// Mitsubishi GX Works2 project: fx3g程序模板   PLC: FX3G

PROGRAM MAIN
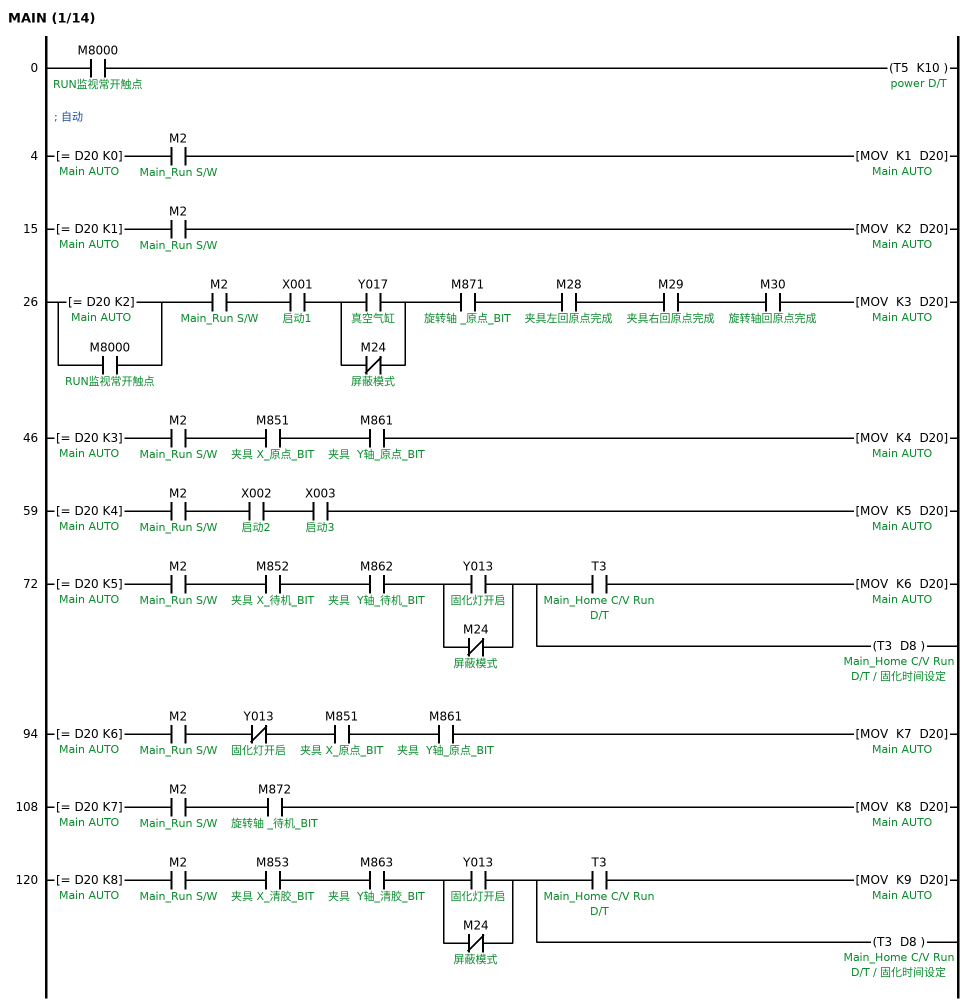
0     LD      M8000  ; RUN监视常开触点
      OUT     T5 K10  ; power D/T
; 自动
4     LD=     D20 K0  ; Main AUTO
      AND     M2  ; Main_Run S/W
      MOV     K1 D20
15    LD=     D20 K1  ; Main AUTO
      AND     M2  ; Main_Run S/W
      MOV     K2 D20
26    LD=     D20 K2  ; Main AUTO
      OR      M8000  ; RUN监视常开触点
      AND     M2  ; Main_Run S/W
      AND     X001  ; 启动1
      LD      Y017  ; 真空气缸
      ORI     M24  ; 屏蔽模式
      ANB
      AND     M871  ; 旋转轴 _原点_BIT
      AND     M28  ; 夹具左回原点完成
      AND     M29  ; 夹具右回原点完成
      AND     M30  ; 旋转轴回原点完成
      MOV     K3 D20
46    LD=     D20 K3  ; Main AUTO
      AND     M2  ; Main_Run S/W
      AND     M851  ; 夹具 X_原点_BIT
      AND     M861  ; 夹具  Y轴_原点_BIT
      MOV     K4 D20
59    LD=     D20 K4  ; Main AUTO
      AND     M2  ; Main_Run S/W
      AND     X002  ; 启动2
      AND     X003  ; 启动3
      MOV     K5 D20
72    LD=     D20 K5  ; Main AUTO
      AND     M2  ; Main_Run S/W
      AND     M852  ; 夹具 X_待机_BIT
      AND     M862  ; 夹具  Y轴_待机_BIT
      LD      Y013  ; 固化灯开启
      ORI     M24  ; 屏蔽模式
      ANB
      MPS
      AND     T3  ; Main_Home C/V Run D/T
      MOV     K6 D20
      MPP
      OUT     T3 D8  ; Main_Home C/V Run D/T / 固化时间设定
94    LD=     D20 K6  ; Main AUTO
      AND     M2  ; Main_Run S/W
      ANI     Y013  ; 固化灯开启
      AND     M851  ; 夹具 X_原点_BIT
      AND     M861  ; 夹具  Y轴_原点_BIT
      MOV     K7 D20
108   LD=     D20 K7  ; Main AUTO
      AND     M2  ; Main_Run S/W
      AND     M872  ; 旋转轴 _待机_BIT
      MOV     K8 D20
120   LD=     D20 K8  ; Main AUTO
      AND     M2  ; Main_Run S/W
      AND     M853  ; 夹具 X_清胶_BIT
      AND     M863  ; 夹具  Y轴_清胶_BIT
      LD      Y013  ; 固化灯开启
      ORI     M24  ; 屏蔽模式
      ANB
      MPS
      AND     T3  ; Main_Home C/V Run D/T
      MOV     K9 D20
      MPP
      OUT     T3 D8  ; Main_Home C/V Run D/T / 固化时间设定
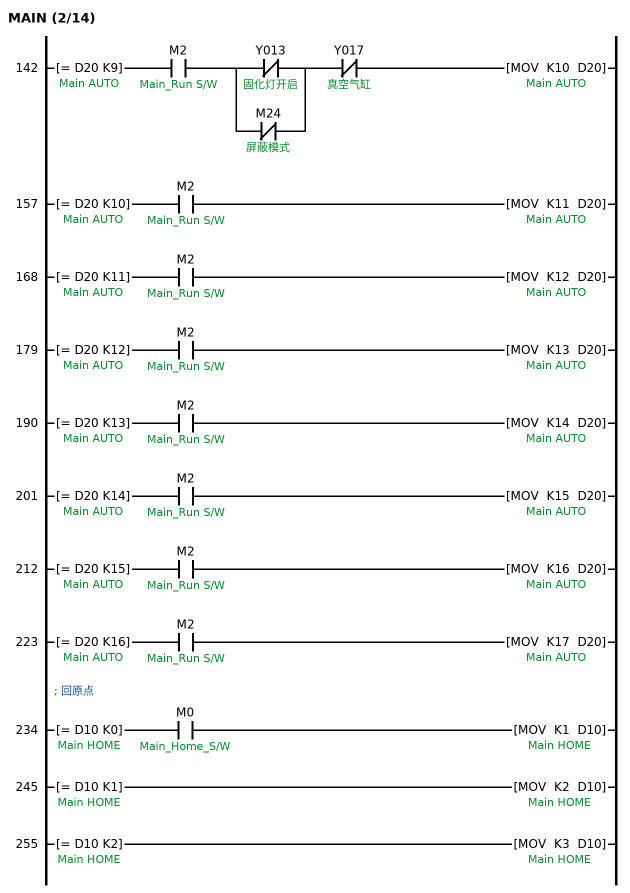
142   LD=     D20 K9  ; Main AUTO
      AND     M2  ; Main_Run S/W
      LDI     Y013  ; 固化灯开启
      ORI     M24  ; 屏蔽模式
      ANB
      ANI     Y017  ; 真空气缸
      MOV     K10 D20
157   LD=     D20 K10  ; Main AUTO
      AND     M2  ; Main_Run S/W
      MOV     K11 D20
168   LD=     D20 K11  ; Main AUTO
      AND     M2  ; Main_Run S/W
      MOV     K12 D20
179   LD=     D20 K12  ; Main AUTO
      AND     M2  ; Main_Run S/W
      MOV     K13 D20
190   LD=     D20 K13  ; Main AUTO
      AND     M2  ; Main_Run S/W
      MOV     K14 D20
201   LD=     D20 K14  ; Main AUTO
      AND     M2  ; Main_Run S/W
      MOV     K15 D20
212   LD=     D20 K15  ; Main AUTO
      AND     M2  ; Main_Run S/W
      MOV     K16 D20
223   LD=     D20 K16  ; Main AUTO
      AND     M2  ; Main_Run S/W
      MOV     K17 D20
; 回原点
234   LD=     D10 K0  ; Main HOME
      AND     M0  ; Main_Home_S/W
      MOV     K1 D10
245   LD=     D10 K1  ; Main HOME
      MOV     K2 D10
255   LD=     D10 K2  ; Main HOME
      MOV     K3 D10
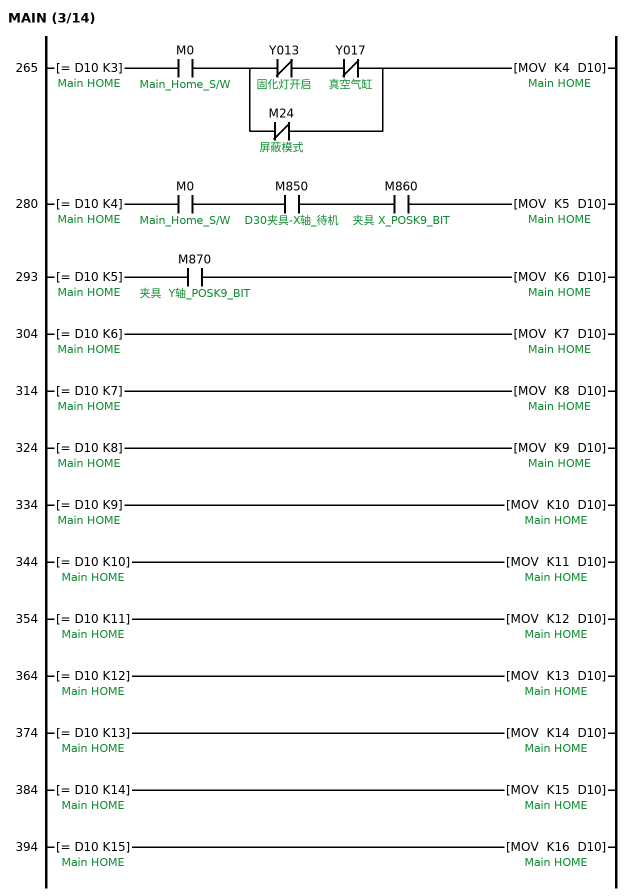
265   LD=     D10 K3  ; Main HOME
      AND     M0  ; Main_Home_S/W
      LDI     Y013  ; 固化灯开启
      ANI     Y017  ; 真空气缸
      ORI     M24  ; 屏蔽模式
      ANB
      MOV     K4 D10
280   LD=     D10 K4  ; Main HOME
      AND     M0  ; Main_Home_S/W
      AND     M850  ; D30夹具-X轴_待机
      AND     M860  ; 夹具 X_POSK9_BIT
      MOV     K5 D10
293   LD=     D10 K5  ; Main HOME
      AND     M870  ; 夹具  Y轴_POSK9_BIT
      MOV     K6 D10
304   LD=     D10 K6  ; Main HOME
      MOV     K7 D10
314   LD=     D10 K7  ; Main HOME
      MOV     K8 D10
324   LD=     D10 K8  ; Main HOME
      MOV     K9 D10
334   LD=     D10 K9  ; Main HOME
      MOV     K10 D10
344   LD=     D10 K10  ; Main HOME
      MOV     K11 D10
354   LD=     D10 K11  ; Main HOME
      MOV     K12 D10
364   LD=     D10 K12  ; Main HOME
      MOV     K13 D10
374   LD=     D10 K13  ; Main HOME
      MOV     K14 D10
384   LD=     D10 K14  ; Main HOME
      MOV     K15 D10
394   LD=     D10 K15  ; Main HOME
      MOV     K16 D10
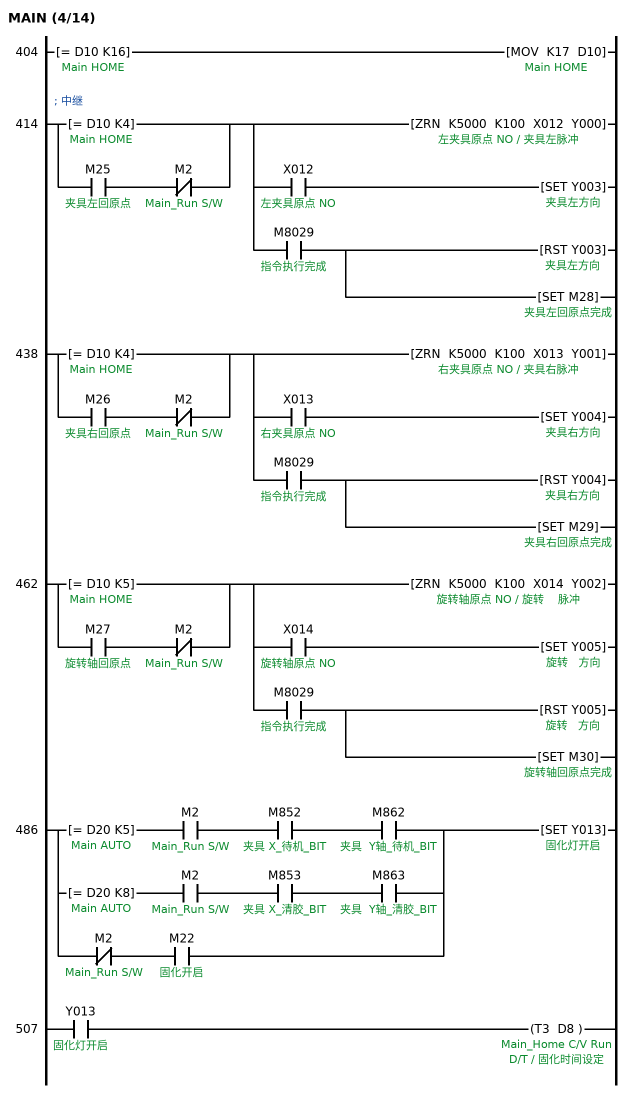
404   LD=     D10 K16  ; Main HOME
      MOV     K17 D10
; 中继
414   LD=     D10 K4  ; Main HOME
      LD      M25  ; 夹具左回原点
      ANI     M2  ; Main_Run S/W
      ORB
      ZRN     K5000 K100 X012 Y000  ; 左夹具原点 NO / 夹具左脉冲
      MPS
      AND     X012  ; 左夹具原点 NO
      SET     Y003  ; 夹具左方向
      MPP
      AND     M8029  ; 指令执行完成
      RST     Y003  ; 夹具左方向
      SET     M28  ; 夹具左回原点完成
438   LD=     D10 K4  ; Main HOME
      LD      M26  ; 夹具右回原点
      ANI     M2  ; Main_Run S/W
      ORB
      ZRN     K5000 K100 X013 Y001  ; 右夹具原点 NO / 夹具右脉冲
      MPS
      AND     X013  ; 右夹具原点 NO
      SET     Y004  ; 夹具右方向
      MPP
      AND     M8029  ; 指令执行完成
      RST     Y004  ; 夹具右方向
      SET     M29  ; 夹具右回原点完成
462   LD=     D10 K5  ; Main HOME
      LD      M27  ; 旋转轴回原点
      ANI     M2  ; Main_Run S/W
      ORB
      ZRN     K5000 K100 X014 Y002  ; 旋转轴原点 NO / 旋转    脉冲
      MPS
      AND     X014  ; 旋转轴原点 NO
      SET     Y005  ; 旋转   方向
      MPP
      AND     M8029  ; 指令执行完成
      RST     Y005  ; 旋转   方向
      SET     M30  ; 旋转轴回原点完成
486   LD=     D20 K5  ; Main AUTO
      AND     M2  ; Main_Run S/W
      AND     M852  ; 夹具 X_待机_BIT
      AND     M862  ; 夹具  Y轴_待机_BIT
      LD=     D20 K8  ; Main AUTO
      AND     M2  ; Main_Run S/W
      AND     M853  ; 夹具 X_清胶_BIT
      AND     M863  ; 夹具  Y轴_清胶_BIT
      ORB
      LDI     M2  ; Main_Run S/W
      AND     M22  ; 固化开启
      ORB
      SET     Y013  ; 固化灯开启
507   LD      Y013  ; 固化灯开启
      OUT     T3 D8  ; Main_Home C/V Run D/T / 固化时间设定
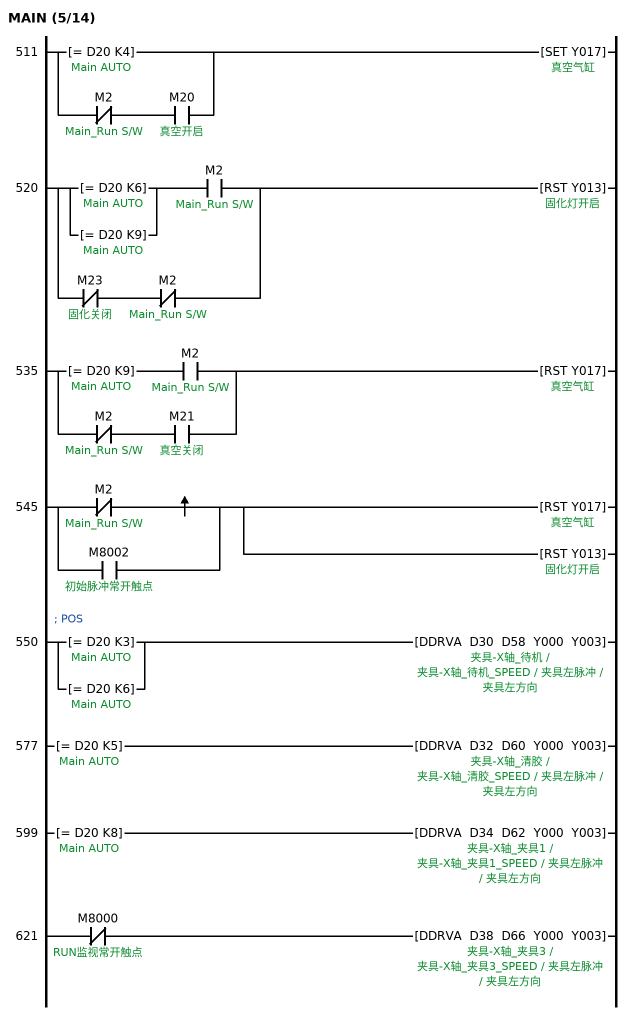
511   LD=     D20 K4  ; Main AUTO
      LDI     M2  ; Main_Run S/W
      AND     M20  ; 真空开启
      ORB
      SET     Y017  ; 真空气缸
520   LD=     D20 K6  ; Main AUTO
      OR=     D20 K9  ; Main AUTO
      AND     M2  ; Main_Run S/W
      LDI     M23  ; 固化关闭
      ANI     M2  ; Main_Run S/W
      ORB
      RST     Y013  ; 固化灯开启
535   LD=     D20 K9  ; Main AUTO
      AND     M2  ; Main_Run S/W
      LDI     M2  ; Main_Run S/W
      AND     M21  ; 真空关闭
      ORB
      RST     Y017  ; 真空气缸
545   LDI     M2  ; Main_Run S/W
      MEP
      OR      M8002  ; 初始脉冲常开触点
      RST     Y017  ; 真空气缸
      RST     Y013  ; 固化灯开启
; POS
550   LD=     D20 K3  ; Main AUTO
      OR=     D20 K6  ; Main AUTO
      DDRVA   D30 D58 Y000 Y003  ; 夹具-X轴_待机 / 夹具-X轴_待机_SPEED
577   LD=     D20 K5  ; Main AUTO
      DDRVA   D32 D60 Y000 Y003  ; 夹具-X轴_清胶 / 夹具-X轴_清胶_SPEED
599   LD=     D20 K8  ; Main AUTO
      DDRVA   D34 D62 Y000 Y003  ; 夹具-X轴_夹具1 / 夹具-X轴_夹具1_SPEED
621   LDI     M8000  ; RUN监视常开触点
      DDRVA   D38 D66 Y000 Y003  ; 夹具-X轴_夹具3 / 夹具-X轴_夹具3_SPEED
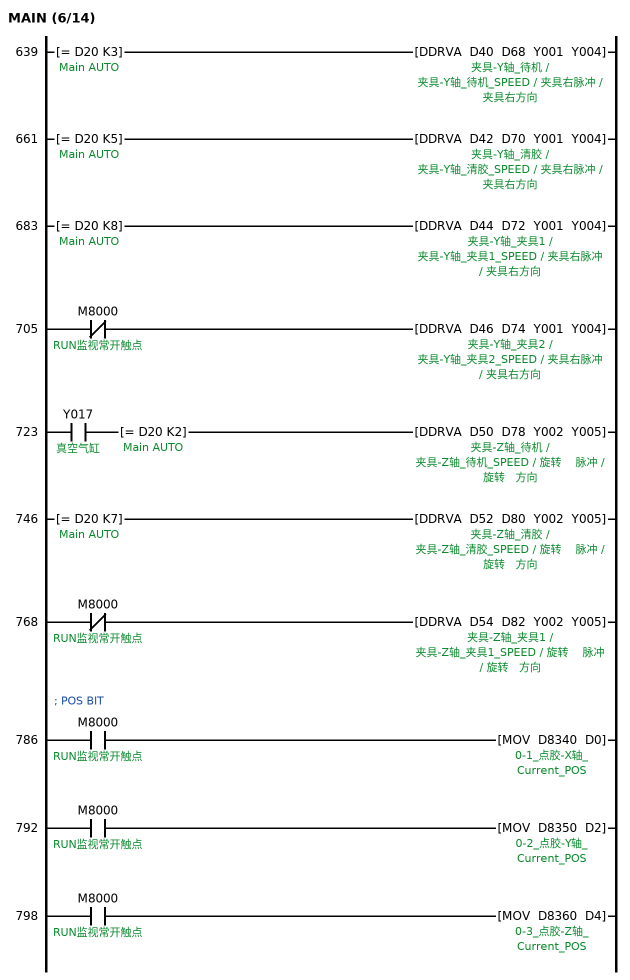
639   LD=     D20 K3  ; Main AUTO
      DDRVA   D40 D68 Y001 Y004  ; 夹具-Y轴_待机 / 夹具-Y轴_待机_SPEED
661   LD=     D20 K5  ; Main AUTO
      DDRVA   D42 D70 Y001 Y004  ; 夹具-Y轴_清胶 / 夹具-Y轴_清胶_SPEED
683   LD=     D20 K8  ; Main AUTO
      DDRVA   D44 D72 Y001 Y004  ; 夹具-Y轴_夹具1 / 夹具-Y轴_夹具1_SPEED
705   LDI     M8000  ; RUN监视常开触点
      DDRVA   D46 D74 Y001 Y004  ; 夹具-Y轴_夹具2 / 夹具-Y轴_夹具2_SPEED
723   LD      Y017  ; 真空气缸
      AND=    D20 K2  ; Main AUTO
      DDRVA   D50 D78 Y002 Y005  ; 夹具-Z轴_待机 / 夹具-Z轴_待机_SPEED
746   LD=     D20 K7  ; Main AUTO
      DDRVA   D52 D80 Y002 Y005  ; 夹具-Z轴_清胶 / 夹具-Z轴_清胶_SPEED
768   LDI     M8000  ; RUN监视常开触点
      DDRVA   D54 D82 Y002 Y005  ; 夹具-Z轴_夹具1 / 夹具-Z轴_夹具1_SPEED
; POS BIT
786   LD      M8000  ; RUN监视常开触点
      MOV     D8340 D0  ; 0-1_点胶-X轴_Current_POS
792   LD      M8000  ; RUN监视常开触点
      MOV     D8350 D2  ; 0-2_点胶-Y轴_Current_POS
798   LD      M8000  ; RUN监视常开触点
      MOV     D8360 D4  ; 0-3_点胶-Z轴_Current_POS
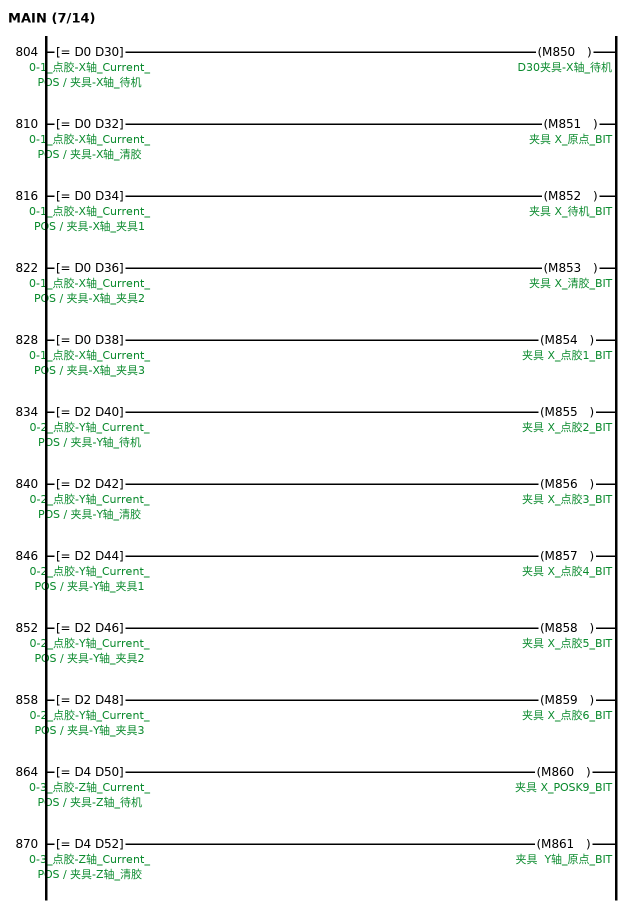
804   LD=     D0 D30  ; 0-1_点胶-X轴_Current_POS / 夹具-X轴_待机
      OUT     M850  ; D30夹具-X轴_待机
810   LD=     D0 D32  ; 0-1_点胶-X轴_Current_POS / 夹具-X轴_清胶
      OUT     M851  ; 夹具 X_原点_BIT
816   LD=     D0 D34  ; 0-1_点胶-X轴_Current_POS / 夹具-X轴_夹具1
      OUT     M852  ; 夹具 X_待机_BIT
822   LD=     D0 D36  ; 0-1_点胶-X轴_Current_POS / 夹具-X轴_夹具2
      OUT     M853  ; 夹具 X_清胶_BIT
828   LD=     D0 D38  ; 0-1_点胶-X轴_Current_POS / 夹具-X轴_夹具3
      OUT     M854  ; 夹具 X_点胶1_BIT
834   LD=     D2 D40  ; 0-2_点胶-Y轴_Current_POS / 夹具-Y轴_待机
      OUT     M855  ; 夹具 X_点胶2_BIT
840   LD=     D2 D42  ; 0-2_点胶-Y轴_Current_POS / 夹具-Y轴_清胶
      OUT     M856  ; 夹具 X_点胶3_BIT
846   LD=     D2 D44  ; 0-2_点胶-Y轴_Current_POS / 夹具-Y轴_夹具1
      OUT     M857  ; 夹具 X_点胶4_BIT
852   LD=     D2 D46  ; 0-2_点胶-Y轴_Current_POS / 夹具-Y轴_夹具2
      OUT     M858  ; 夹具 X_点胶5_BIT
858   LD=     D2 D48  ; 0-2_点胶-Y轴_Current_POS / 夹具-Y轴_夹具3
      OUT     M859  ; 夹具 X_点胶6_BIT
864   LD=     D4 D50  ; 0-3_点胶-Z轴_Current_POS / 夹具-Z轴_待机
      OUT     M860  ; 夹具 X_POSK9_BIT
870   LD=     D4 D52  ; 0-3_点胶-Z轴_Current_POS / 夹具-Z轴_清胶
      OUT     M861  ; 夹具  Y轴_原点_BIT
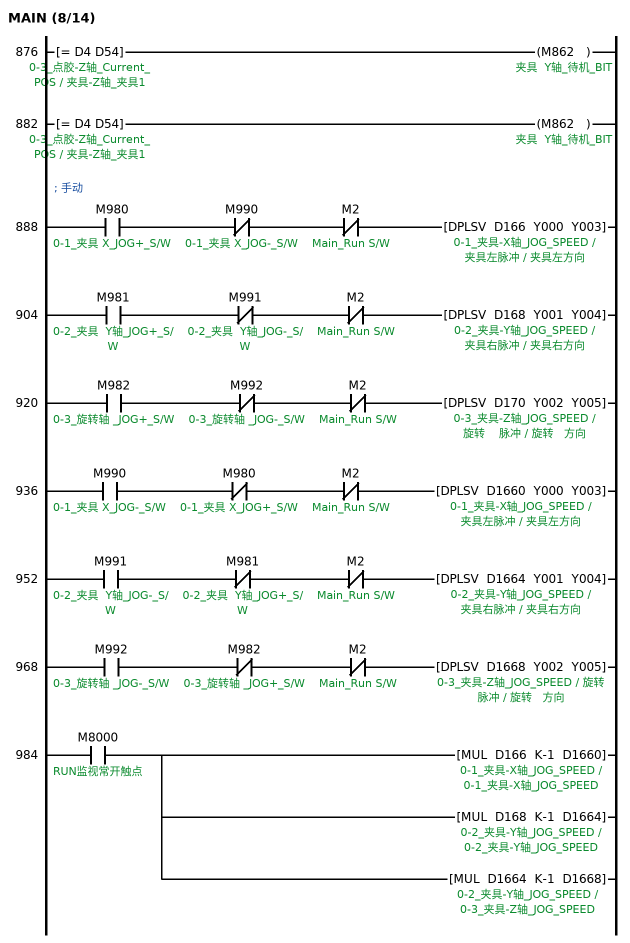
876   LD=     D4 D54  ; 0-3_点胶-Z轴_Current_POS / 夹具-Z轴_夹具1
      OUT     M862  ; 夹具  Y轴_待机_BIT
882   LD=     D4 D54  ; 0-3_点胶-Z轴_Current_POS / 夹具-Z轴_夹具1
      OUT     M862  ; 夹具  Y轴_待机_BIT
; 手动
888   LD      M980  ; 0-1_夹具 X_JOG+_S/W
      ANI     M990  ; 0-1_夹具 X_JOG-_S/W
      ANI     M2  ; Main_Run S/W
      DPLSV   D166 Y000 Y003  ; 0-1_夹具-X轴_JOG_SPEED
904   LD      M981  ; 0-2_夹具  Y轴_JOG+_S/W
      ANI     M991  ; 0-2_夹具  Y轴_JOG-_S/W
      ANI     M2  ; Main_Run S/W
      DPLSV   D168 Y001 Y004  ; 0-2_夹具-Y轴_JOG_SPEED
920   LD      M982  ; 0-3_旋转轴 _JOG+_S/W
      ANI     M992  ; 0-3_旋转轴 _JOG-_S/W
      ANI     M2  ; Main_Run S/W
      DPLSV   D170 Y002 Y005  ; 0-3_夹具-Z轴_JOG_SPEED
936   LD      M990  ; 0-1_夹具 X_JOG-_S/W
      ANI     M980  ; 0-1_夹具 X_JOG+_S/W
      ANI     M2  ; Main_Run S/W
      DPLSV   D1660 Y000 Y003  ; 0-1_夹具-X轴_JOG_SPEED
952   LD      M991  ; 0-2_夹具  Y轴_JOG-_S/W
      ANI     M981  ; 0-2_夹具  Y轴_JOG+_S/W
      ANI     M2  ; Main_Run S/W
      DPLSV   D1664 Y001 Y004  ; 0-2_夹具-Y轴_JOG_SPEED
968   LD      M992  ; 0-3_旋转轴 _JOG-_S/W
      ANI     M982  ; 0-3_旋转轴 _JOG+_S/W
      ANI     M2  ; Main_Run S/W
      DPLSV   D1668 Y002 Y005  ; 0-3_夹具-Z轴_JOG_SPEED
984   LD      M8000  ; RUN监视常开触点
      MUL     D166 K-1 D1660
      MUL     D168 K-1 D1664
      MUL     D1664 K-1 D1668
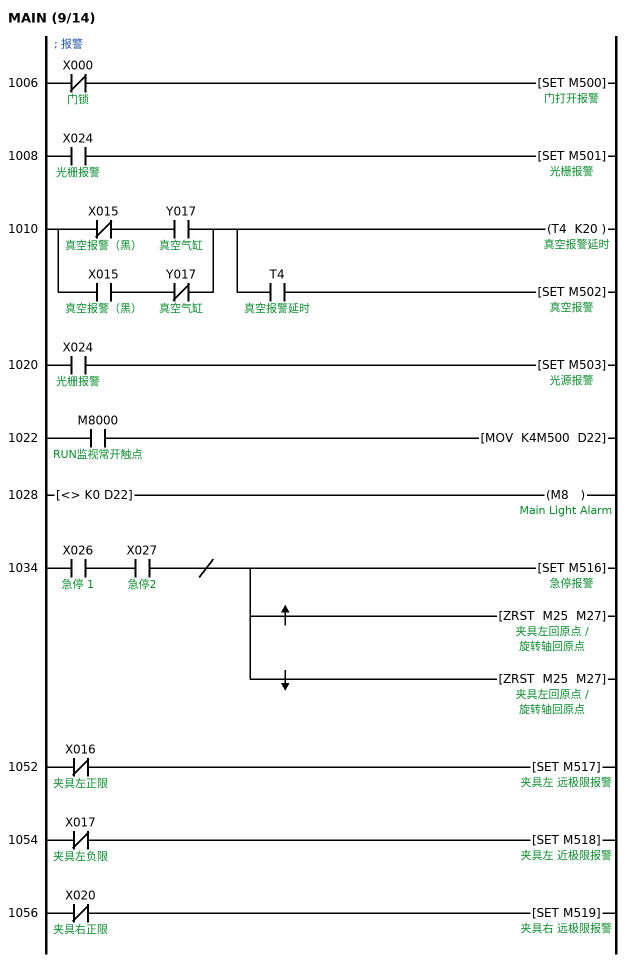
; 报警
1006  LDI     X000  ; 门锁
      SET     M500  ; 门打开报警
1008  LD      X024  ; 光栅报警
      SET     M501  ; 光栅报警
1010  LDI     X015  ; 真空报警（黑）
      AND     Y017  ; 真空气缸
      LD      X015  ; 真空报警（黑）
      ANI     Y017  ; 真空气缸
      ORB
      OUT     T4 K20  ; 真空报警延时
      AND     T4  ; 真空报警延时
      SET     M502  ; 真空报警
1020  LD      X024  ; 光栅报警
      SET     M503  ; 光源报警
1022  LD      M8000  ; RUN监视常开触点
      MOV     K4M500 D22
1028  LD<>    K0 D22
      OUT     M8  ; Main Light Alarm
1034  LD      X026  ; 急停 1
      AND     X027  ; 急停2
      INV
      SET     M516  ; 急停报警
      MPS
      MEP
      ZRST    M25 M27
      MPP
      MEF
      ZRST    M25 M27
1052  LDI     X016  ; 夹具左正限
      SET     M517  ; 夹具左 远极限报警
1054  LDI     X017  ; 夹具左负限
      SET     M518  ; 夹具左 近极限报警
1056  LDI     X020  ; 夹具右正限
      SET     M519  ; 夹具右 远极限报警
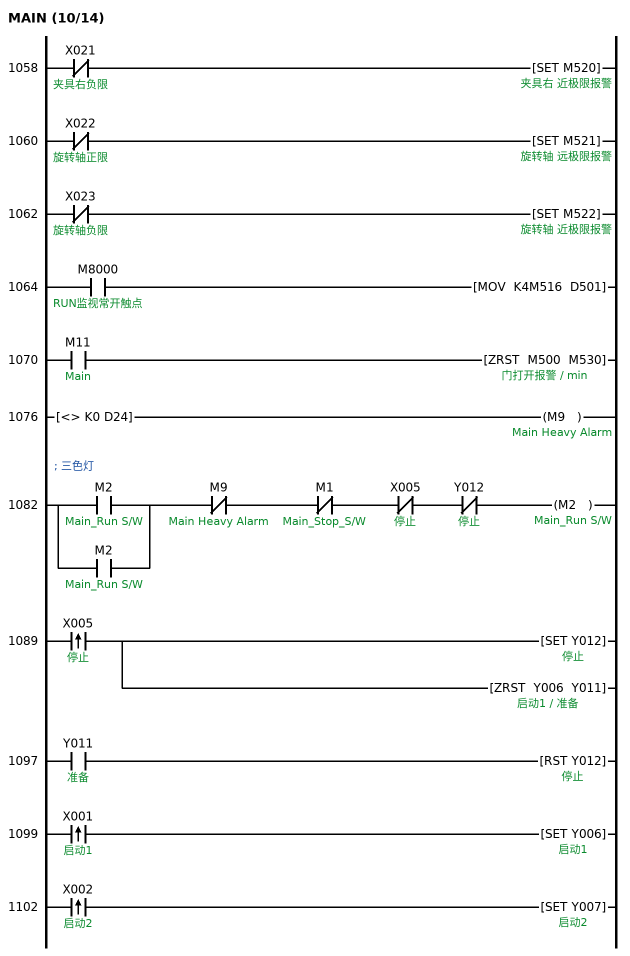
1058  LDI     X021  ; 夹具右负限
      SET     M520  ; 夹具右 近极限报警
1060  LDI     X022  ; 旋转轴正限
      SET     M521  ; 旋转轴 远极限报警
1062  LDI     X023  ; 旋转轴负限
      SET     M522  ; 旋转轴 近极限报警
1064  LD      M8000  ; RUN监视常开触点
      MOV     K4M516 D501
1070  LD      M11  ; Main
      ZRST    M500 M530  ; min
1076  LD<>    K0 D24
      OUT     M9  ; Main Heavy Alarm
; 三色灯
1082  LD      M2  ; Main_Run S/W
      OR      M2  ; Main_Run S/W
      ANI     M9  ; Main Heavy Alarm
      ANI     M1  ; Main_Stop_S/W
      ANI     X005  ; 停止
      ANI     Y012  ; 停止
      OUT     M2  ; Main_Run S/W
1089  LDP     X005  ; 停止
      SET     Y012  ; 停止
      ZRST    Y006 Y011  ; 启动1 / 准备
1097  LD      Y011  ; 准备
      RST     Y012  ; 停止
1099  LDP     X001  ; 启动1
      SET     Y006  ; 启动1
1102  LDP     X002  ; 启动2
      SET     Y007  ; 启动2
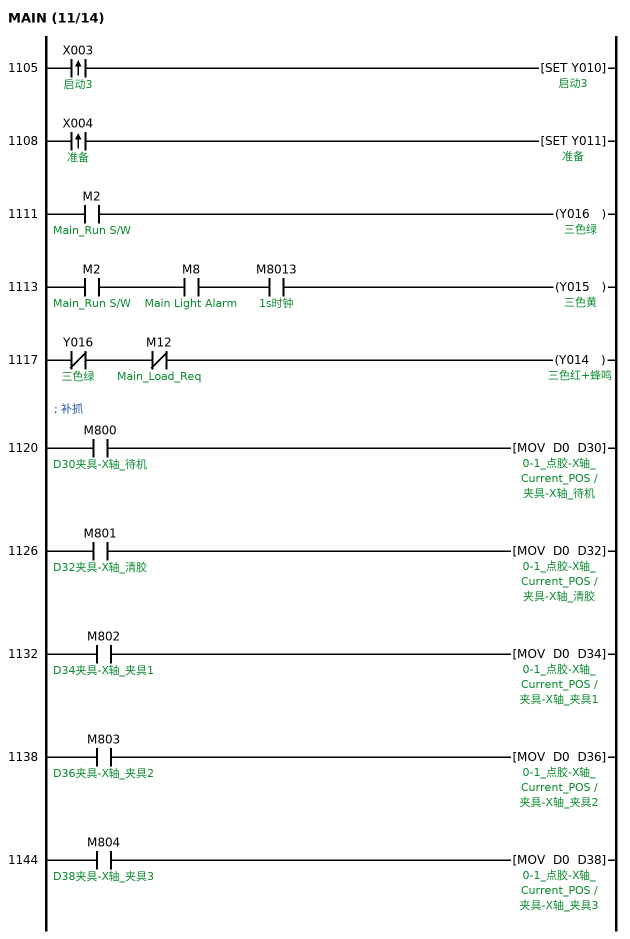
1105  LDP     X003  ; 启动3
      SET     Y010  ; 启动3
1108  LDP     X004  ; 准备
      SET     Y011  ; 准备
1111  LD      M2  ; Main_Run S/W
      OUT     Y016  ; 三色绿
1113  LD      M2  ; Main_Run S/W
      AND     M8  ; Main Light Alarm
      AND     M8013  ; 1s时钟
      OUT     Y015  ; 三色黄
1117  LDI     Y016  ; 三色绿
      ANI     M12  ; Main_Load_Req
      OUT     Y014  ; 三色红+蜂鸣
; 补抓
1120  LD      M800  ; D30夹具-X轴_待机
      MOV     D0 D30
1126  LD      M801  ; D32夹具-X轴_清胶
      MOV     D0 D32
1132  LD      M802  ; D34夹具-X轴_夹具1
      MOV     D0 D34
1138  LD      M803  ; D36夹具-X轴_夹具2
      MOV     D0 D36
1144  LD      M804  ; D38夹具-X轴_夹具3
      MOV     D0 D38
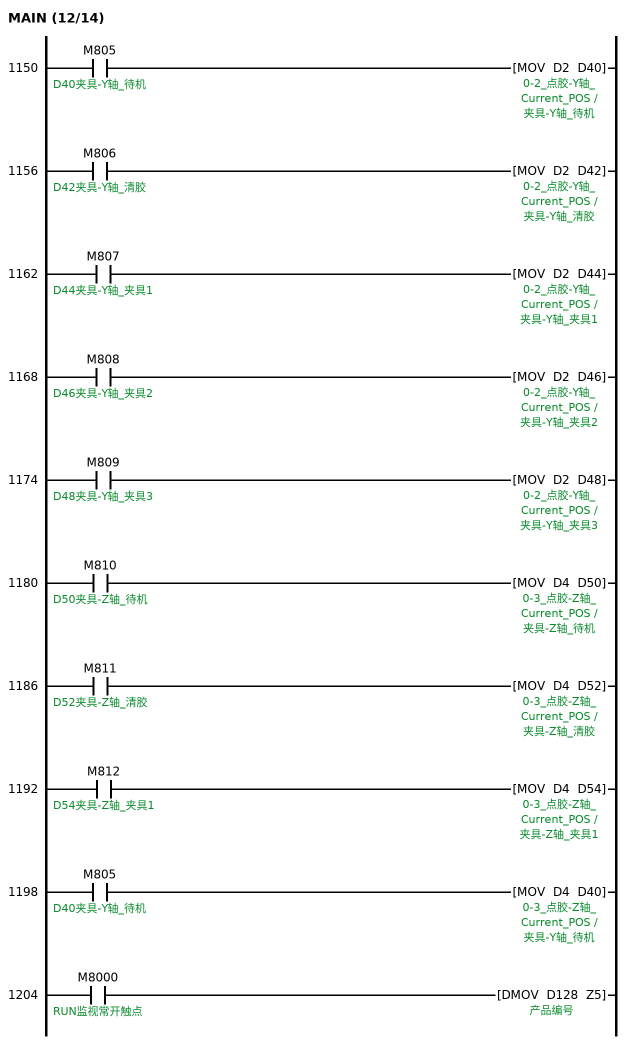
1150  LD      M805  ; D40夹具-Y轴_待机
      MOV     D2 D40
1156  LD      M806  ; D42夹具-Y轴_清胶
      MOV     D2 D42
1162  LD      M807  ; D44夹具-Y轴_夹具1
      MOV     D2 D44
1168  LD      M808  ; D46夹具-Y轴_夹具2
      MOV     D2 D46
1174  LD      M809  ; D48夹具-Y轴_夹具3
      MOV     D2 D48
1180  LD      M810  ; D50夹具-Z轴_待机
      MOV     D4 D50
1186  LD      M811  ; D52夹具-Z轴_清胶
      MOV     D4 D52
1192  LD      M812  ; D54夹具-Z轴_夹具1
      MOV     D4 D54
1198  LD      M805  ; D40夹具-Y轴_待机
      MOV     D4 D40
1204  LD      M8000  ; RUN监视常开触点
      DMOV    D128 Z5  ; 产品编号
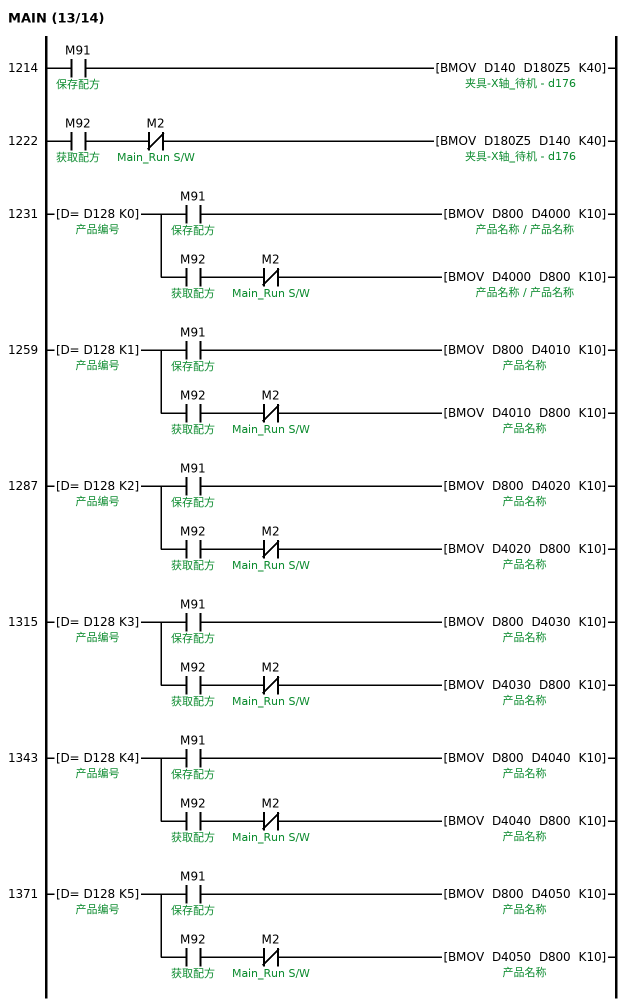
1214  LD      M91  ; 保存配方
      BMOV    D140 D180Z5 K40  ; 夹具-X轴_待机 - d176
1222  LD      M92  ; 获取配方
      ANI     M2  ; Main_Run S/W
      BMOV    D180Z5 D140 K40
1231  LDD=    D128 K0  ; 产品编号
      MPS
      AND     M91  ; 保存配方
      BMOV    D800 D4000 K10  ; 产品名称 / 产品名称
      MPP
      AND     M92  ; 获取配方
      ANI     M2  ; Main_Run S/W
      BMOV    D4000 D800 K10
1259  LDD=    D128 K1  ; 产品编号
      MPS
      AND     M91  ; 保存配方
      BMOV    D800 D4010 K10
      MPP
      AND     M92  ; 获取配方
      ANI     M2  ; Main_Run S/W
      BMOV    D4010 D800 K10
1287  LDD=    D128 K2  ; 产品编号
      MPS
      AND     M91  ; 保存配方
      BMOV    D800 D4020 K10
      MPP
      AND     M92  ; 获取配方
      ANI     M2  ; Main_Run S/W
      BMOV    D4020 D800 K10
1315  LDD=    D128 K3  ; 产品编号
      MPS
      AND     M91  ; 保存配方
      BMOV    D800 D4030 K10
      MPP
      AND     M92  ; 获取配方
      ANI     M2  ; Main_Run S/W
      BMOV    D4030 D800 K10
1343  LDD=    D128 K4  ; 产品编号
      MPS
      AND     M91  ; 保存配方
      BMOV    D800 D4040 K10
      MPP
      AND     M92  ; 获取配方
      ANI     M2  ; Main_Run S/W
      BMOV    D4040 D800 K10
1371  LDD=    D128 K5  ; 产品编号
      MPS
      AND     M91  ; 保存配方
      BMOV    D800 D4050 K10
      MPP
      AND     M92  ; 获取配方
      ANI     M2  ; Main_Run S/W
      BMOV    D4050 D800 K10
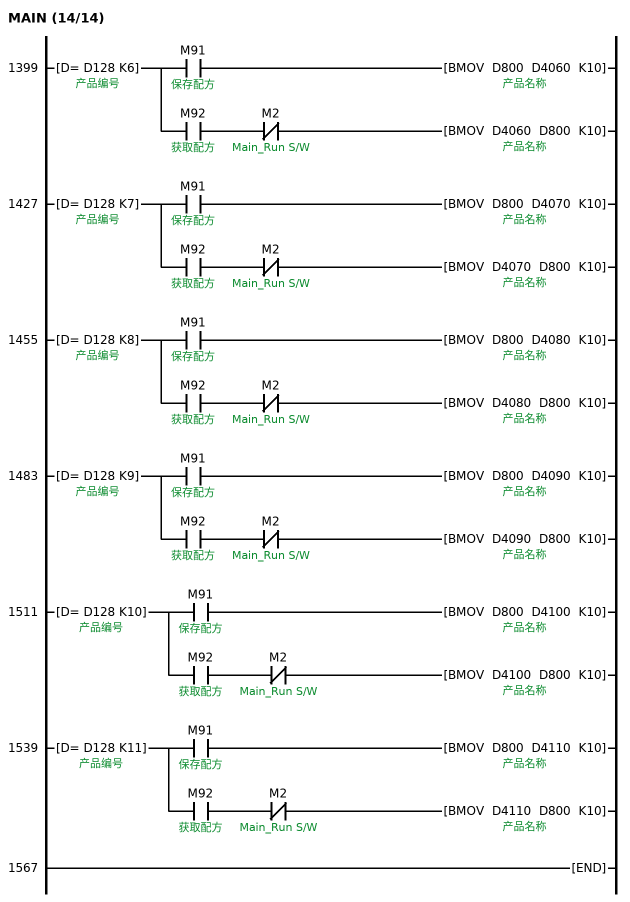
1399  LDD=    D128 K6  ; 产品编号
      MPS
      AND     M91  ; 保存配方
      BMOV    D800 D4060 K10
      MPP
      AND     M92  ; 获取配方
      ANI     M2  ; Main_Run S/W
      BMOV    D4060 D800 K10
1427  LDD=    D128 K7  ; 产品编号
      MPS
      AND     M91  ; 保存配方
      BMOV    D800 D4070 K10
      MPP
      AND     M92  ; 获取配方
      ANI     M2  ; Main_Run S/W
      BMOV    D4070 D800 K10
1455  LDD=    D128 K8  ; 产品编号
      MPS
      AND     M91  ; 保存配方
      BMOV    D800 D4080 K10
      MPP
      AND     M92  ; 获取配方
      ANI     M2  ; Main_Run S/W
      BMOV    D4080 D800 K10
1483  LDD=    D128 K9  ; 产品编号
      MPS
      AND     M91  ; 保存配方
      BMOV    D800 D4090 K10
      MPP
      AND     M92  ; 获取配方
      ANI     M2  ; Main_Run S/W
      BMOV    D4090 D800 K10
1511  LDD=    D128 K10  ; 产品编号
      MPS
      AND     M91  ; 保存配方
      BMOV    D800 D4100 K10
      MPP
      AND     M92  ; 获取配方
      ANI     M2  ; Main_Run S/W
      BMOV    D4100 D800 K10
1539  LDD=    D128 K11  ; 产品编号
      MPS
      AND     M91  ; 保存配方
      BMOV    D800 D4110 K10
      MPP
      AND     M92  ; 获取配方
      ANI     M2  ; Main_Run S/W
      BMOV    D4110 D800 K10
1567  END
END_PROGRAM

// device comments not shown above
X025  ; 光源报警
M3  ; Main_Alarm
M4  ; Main_PNL_Exist
M5  ; Main_PNL_Arrived
M6  ; Main_PNL_Leaving
M7  ; Main_Axis Home NG
M10  ; Main_PNL_NG
M13  ; Main_Load_Comp
M14  ; Main_Unload_Req
M15  ; Main_Unload_Comp
M700  ; 夹具 X_原点_S/W
M701  ; 夹具 X_待机_S/W
M702  ; 夹具 X_清胶_S/W
M703  ; 夹具 X_点胶1_S/W
M704  ; 夹具 X_点胶2_S/W
M705  ; 夹具 X_点胶3_S/W
M706  ; 夹具 X_点胶4_S/W
M707  ; 夹具 X_点胶5_S/W
M708  ; 夹具 X_点胶6_S/W
M709  ; 夹具 X_POSK9_S/W
M710  ; 夹具  Y轴_原点_S/W
M711  ; 夹具  Y轴_待机_S/W
M712  ; 夹具  Y轴_清胶_S/W
M713  ; 夹具  Y轴_点胶1_S/W
M714  ; 夹具  Y轴_点胶2_S/W
M715  ; 夹具  Y轴_点胶3_S/W
M716  ; 夹具  Y轴_点胶4_S/W
M717  ; 夹具  Y轴_点胶5_S/W
M718  ; 夹具  Y轴_点胶6_S/W
M719  ; 夹具  Y轴_POSK9_S/W
M720  ; 旋转轴
M721  ; 旋转轴 _待机_S/W
M722  ; 旋转轴 _清胶_S/W
M750  ; 夹具 X_原点_Trig
M751  ; 夹具 X_待机_Trig
M752  ; 夹具 X_清胶_Trig
M753  ; 夹具 X_点胶1_Trig
M754  ; 夹具 X_点胶2_Trig
M755  ; 夹具 X_点胶3_Trig
M756  ; 夹具 X_点胶4_Trig
M757  ; 夹具 X_点胶5_Trig
M758  ; 夹具 X_点胶6_Trig
M759  ; 夹具 X_POSK9_Trig
M760  ; 夹具  Y轴_原点_Trig
M761  ; 夹具  Y轴_待机_Trig
M762  ; 夹具  Y轴_清胶_Trig
M763  ; 夹具  Y轴_点胶1_Trig
M764  ; 夹具  Y轴_点胶2_Trig
M765  ; 夹具  Y轴_点胶3_Trig
M766  ; 夹具  Y轴_点胶4_Trig
M767  ; 夹具  Y轴_点胶5_Trig
M768  ; 夹具  Y轴_点胶6_Trig
M769  ; 夹具  Y轴_POSK9_Trig
M770  ; 旋转轴 _原点_Trig
M771  ; 旋转轴 _待机_Trig
M772  ; 旋转轴 _清胶_Trig
M864  ; 夹具  Y轴_点胶1_BIT
M865  ; 夹具  Y轴_点胶2_BIT
M866  ; 夹具  Y轴_点胶3_BIT
M867  ; 夹具  Y轴_点胶4_BIT
M868  ; 夹具  Y轴_点胶5_BIT
M869  ; 夹具  Y轴_点胶6_BIT
M873  ; 旋转轴 _清胶_BIT
M880  ; ALL HOME OK BIT
M881  ; ALL STOP  BIT
M884  ; 1.Standby
M885  ; 2.Run
M886  ; 3.Down
M887  ; 4.Error
M888  ; CIM_ONLINE
M889  ; CIM_OFFLINE
M890  ; AUTO MODE
M891  ; MANUAL MODE
M892  ; ALL AUTO RUN
M893  ; ALL RUN BIT
M900  ; 夹具 X_原点_Condition
M901  ; 夹具 X_待机_Condition
M902  ; 夹具 X_清胶_Condition
M903  ; 夹具 X_点胶1_Condition
M904  ; 夹具 X_点胶2_Condition
M905  ; 夹具 X_点胶3_Condition
M906  ; 夹具 X_点胶4_Condition
M907  ; 夹具 X_点胶5_Condition
M908  ; 夹具 X_点胶6_Condition
M909  ; 夹具 X_POSK9_Condition
M910  ; 夹具  Y轴_原点_Condition
M911  ; 夹具  Y轴_待机_Condition
M912  ; 夹具  Y轴_清胶_Condition
M913  ; 夹具  Y轴_点胶1_Condition
M914  ; 夹具  Y轴_点胶2_Condition
M915  ; 夹具  Y轴_点胶3_Condition
M916  ; 夹具  Y轴_点胶4_Condition
M917  ; 夹具  Y轴_点胶5_Condition
M918  ; 夹具  Y轴_点胶6_Condition
M919  ; 夹具  Y轴_POSK9_Condition
M920  ; 旋转轴 _原点_Condition
M921  ; 旋转轴 _待机_Condition
M922  ; 旋转轴 _清胶_Condition
M923  ; 旋转轴 _点胶1_Condition
M924  ; 旋转轴 _点胶2_Condition
M925  ; 旋转轴 _点胶3_Condition
M926  ; 旋转轴 _点胶4_Condition
M927  ; 旋转轴 _点胶5_Condition
M928  ; 旋转轴 _点胶6_Condition
M929  ; 旋转轴 _POSK9_Condition
M930  ; 清胶-Q轴_原点_Condition
M931  ; 清胶-Q轴_POSK1_Condition
M950  ; 0-1_夹具 X Power_Off_S/W
M951  ; 0-2_夹具  Y轴 Power_Off_S/W
M952  ; 0-3_旋转轴  Power_Off_S/W
M953  ; 0-4_清胶-Q轴 Power_Off_S/W
M960  ; 0-1_夹具 XPower_Off_Trig
M961  ; 0-2_夹具  Y轴Power_Off_Trig
M962  ; 0-3_旋转轴 Power_Off_Trig
M963  ; 0-4_清胶-Q轴Power_Off_Trig
M970  ; 0-1_夹具 X SERVO
M971  ; 0-2_夹具  Y轴 SERVO
M972  ; 0-3_旋转轴  SERVO
M973  ; 0-4_清胶-Q轴 SERVO
M983  ; 0-4_清胶-Q轴_JOG+_S/W
M993  ; 0-4_清胶-Q轴_JOG-_S/W
M1020  ; 0-1_夹具 X Home_OK_Keep
M1021  ; 0-2_夹具  Y轴 Home_OK_Keep
M1022  ; 0-3_旋转轴  Home_OK_Keep
M1023  ; 0-4_清胶-Q轴 Home_OK_Keep
M1080  ; All_Home_S/W
M1081  ; All Stop S/W
M1082  ; All_Home_TRIG
M1083  ; All Stop TRIG
M1090  ; AUTO MODE S/W
M1091  ; MANUAL MODE S/W
M1100  ; ALL RUN TRIG
M1101  ; ALL RUN S/W
M1102  ; ALL_START_S/W_TRIG
M1104  ; ALL_TR_STOP_TRIG
M1110  ; ALARM  RESET S/W
M1111  ; ALARM RESET BIT
M1112  ; Buzer Stop S/W
M1118  ; EMG STOP CHECK NG
M1120  ; EMG STOP CHECK OK
M1121  ; DOOR CLOSE OK
M1122  ; DOOR_PASS S/W
M1130  ; PNL SUPPLY STOP
M1131  ; PNL SUPPLY 1 SHEET
M1132  ; POS_Auto_Calculate_S/W
M1140  ; TOUCH_ACC/DEC
M1141  ; TOUCH_POS_SETTING
M1142  ; TOUCH_MANUAL
M1143  ; TOUCH_SERVO_TOURQUE
M1144  ; TOUCH_HOME_DFFSET
M1170  ; QD_POS_SPEED_TRANSFER
M1172  ; QD77-1_READY_RETRY
M1173  ; QD77-2_READY_RETRY
M1178  ; MACHINE ALARM
M1179  ; SYSTEM ALARM
M1510  ; Recipe Save OK Button
M1511  ; Recipe Save Ok Trig
M1512  ; Recipe Buffer Area Write Comp
M1515  ; Recipe Save Interlock
M1525  ; RECIPE BODY INTERLOCK BIT
M1526  ; Recipe Body Select Bit
M1530  ; Recipe Copy Button
M1535  ; Recipe Copy Interlock
M1540  ; Recipe Copy Source Up
M1541  ; Recipe Copy Source Down
M1542  ; Recipe Copy Target Up
M1543  ; Recipe Copy Target Down
M1550  ; Recipe Change Button
M1555  ; Recipe Change Interlock
M1560  ; Recipe Change No Up
M1561  ; Recipe Change No Down
D12  ; 型号显示
D64  ; 夹具-X轴_夹具2_SPEED
D76  ; 夹具-Y轴_夹具3_SPEED
D142  ; 夹具-X轴_清胶
D144  ; 夹具-X轴_夹具1
D146  ; 夹具-X轴_夹具2
D148  ; 夹具-X轴_夹具3
D150  ; 夹具-Y轴_待机
D152  ; 夹具-Y轴_清胶
D154  ; 夹具-Y轴_夹具1
D156  ; 夹具-Y轴_夹具2
D158  ; 夹具-Y轴_夹具3
D160  ; 夹具-Z轴_待机
D162  ; 夹具-Z轴_清胶
D164  ; 夹具-Z轴_夹具1
D172  ; 0-1_夹具-X轴_ACC/DEC_TIME
D174  ; 0-2_夹具-Y轴_ACC/DEC_TIME
D176  ; 0-3_夹具-Z轴_ACC/DEC_TIME
D180  ; D180
D204  ; D204
D228  ; D228
D252  ; D252
D276  ; D276
D300  ; D300
D324  ; D324
D348  ; D348
D372  ; D372
D396  ; D396
D420  ; D420
D444  ; D444
D468  ; D468
D492  ; D492
D516  ; D516
D540  ; D540
D564  ; D564
D588  ; D588
D612  ; D612
D636  ; D636
D660  ; D660
D684  ; D684
D708  ; D708
D732  ; D732
D756  ; D756
D780  ; D780
D804  ; D804
D828  ; D828
D852  ; D852
D876  ; D876
D900  ; D900
D924  ; D924
D948  ; D948
T0  ; Main_Home Trig D/T
T1  ; Main_Force Stop D/T
T2  ; Main_Home Step D/T
T100  ; 0-1_点胶-X轴 Busy_Off_D/T
T101  ; 0-2_点胶-Y轴 Busy_Off_D/T
T102  ; 0-3_点胶-Z轴 Busy_Off_D/T
T103  ; 0-4_清胶-Q轴 Busy_Off_D/T
T200  ; AUTO_RUN_D/T
T202  ; POWER ON D/T
T203  ; QD77_POWER_ON_D/T
T204  ; QD_POS_SPEED_TRANSFER_COMP
T205  ; RECIPE SAVE D/T
T206  ; Recipe Change Delaytime
T207  ; Recipe Copy Delaytime
T208  ; RECIPE DELETE D/T
T209  ; RECIPE NAME CHANGE D/T
